// TIA Portal V19 export
DATA_BLOCK "PPrgArchive16"   // DB504
// stored: IsOnlyStoredInLoadMemory true, MemoryReserve 0, Namespace G
   VAR RETAIN
      PRG : Array[1501..1600] of "PPrg_Data";
   END_VAR
BEGIN
END_DATA_BLOCK
